Yaskawa INFORM job: MAT.JBI

/JOB
//NAME MAT
//POS
///NPOS 2,0,0,0,0,0
///TOOL 0
///POSTYPE PULSE
///PULSE
C00000=160456,-29023,168816,-9259,-120073,14761
C00001=90155,-10653,158157,-9260,-120074,14760
//INST
///DATE 2018/08/06 09:48
///ATTR SC,RW
///GROUP1 RB1
NOP
MOVJ C00000 VJ=15.00
MOVL C00001 V=150.0
END
